DATA_BLOCK "ST10_Stopper_FB_DB"
VAR
  FB_Stopper_Instance : Array[1..3] of "FB_Stopper";
END_VAR
BEGIN
END_DATA_BLOCK
